FUNCTION_BLOCK OperationStatus (* Basic Function Block Type *)
  (* Standard: 61499-2 *)
  (* Version 0.0, 11/3/2020, prana, nxtControl GmbH, Template *)
  PACKAGE Main;
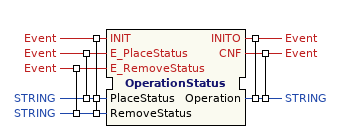
  EVENT_INPUT
    INIT WITH PlaceStatus, RemoveStatus; (* Initialization Request *)
    E_PlaceStatus WITH PlaceStatus; (* Normal Execution Request *)
    E_RemoveStatus WITH RemoveStatus;
  END_EVENT
  EVENT_OUTPUT
    INITO WITH Operation; (* Initialization Confirm *)
    CNF WITH Operation; (* Execution Confirmation *)
  END_EVENT
  VAR_INPUT
    PlaceStatus : STRING; (* Input event qualifier *)
    RemoveStatus : STRING;
  END_VAR
  VAR_OUTPUT
    Operation : STRING; (* Output event qualifier *)
  END_VAR
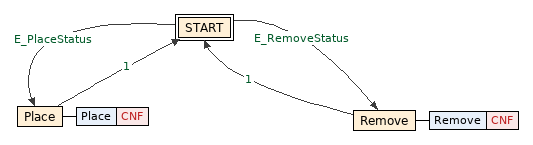
  EC_STATES
    START; (* Initial State *)
    Place : Place -> CNF;
    Remove : Remove -> CNF;
  END_STATES
  EC_TRANSITIONS
    START TO Place := E_PlaceStatus;
    START TO Remove := E_RemoveStatus;
    Remove TO START := 1;
    Place TO START := 1;
  END_TRANSITIONS
  ALGORITHM Place IN ST: (* Initialization algorithm *)
Operation := CONCAT('P',PlaceStatus);
  END_ALGORITHM
  ALGORITHM Remove IN ST: (* Normally executed algorithm *)
Operation := CONCAT('R',RemoveStatus);
  END_ALGORITHM
END_FUNCTION_BLOCK
